// TIA Portal project "TankFillingSystem_V16" (V16)

(* hardware
DEVICE "S71500/ET200MP station_1"  S7-1500 station
   slot 0: "Rail_0"  Rack  6ES7 590-1***0-0AA0
   slot 1: "Tank filling controller"  CPU 1511C-1 PN  6ES7 511-1CK01-0AB0  V2.8
      slot 3: "CPU display_1"  6ES7591-1AA00-0AA0
      slot 32768: "PROFINET interface_1"  X1
         slot 32769: "Port_1"  X1 P1
         slot 32770: "Port_2"  X1 P2
      slot 34817: "Virtual CP interface port_1"  Virtual CP interface port  Virtual CP interface port
*)

// ===== PLC "Tank filling controller"  CPU 1511C-1 PN =====

VAR_GLOBAL   // PLC tag table "Default tag table"
   "Manual_Start" AT %I0.0 : Bool;
   "Work" AT %M2.0 : Bool;
   "Low_Level_Sensor" AT %I0.1 : Bool;
   "Low_Level" AT %M2.1 : Bool;
   "High_Level" AT %M2.2 : Bool;
   "Top_Level_Sensor" AT %I0.2 : Bool;
   "Manual_Stop" AT %I0.7 : Bool;
   "Manual_Valve_Control" AT %I0.3 : Bool;
   "Valve_Open" AT %M2.3 : Bool;
   "Tag_1" AT %I1.1 : Bool;
   "Manual_Confirm" AT %I0.6 : Bool;
   "Confirm" AT %M2.4 : Bool;
   "Clock_Byte" AT %MB50 : Byte;
   "Clock_10Hz" AT %M50.0 : Bool;
   "Clock_5Hz" AT %M50.1 : Bool;
   "Clock_2.5Hz" AT %M50.2 : Bool;
   "Clock_2Hz" AT %M50.3 : Bool;
   "Clock_1.25Hz" AT %M50.4 : Bool;
   "Clock_1Hz" AT %M50.5 : Bool;
   "Clock_0.625Hz" AT %M50.6 : Bool;
   "Clock_0.5Hz" AT %M50.7 : Bool;
   "Liquid_Montion_Sim" AT %M30.0 : Bool;
   "Emergency_Channel_Gen_Edge" AT %M2.5 : Bool;
   "Malfunction_Memory" AT %M2.6 : Bool;
   "Emergency_Channel_Malfunction_Edge" AT %M2.7 : Bool;
END_VAR

DATA_BLOCK "Tank1_DB"   // DB1
{ S7_Optimized_Access := 'TRUE' }
VERSION : 0.1
// stored: InstanceOfName Tank
"Tank"
BEGIN
   Capacity := 1000.0;
   Fill_Level := 1000.0;
   Growth := 2.5;
END_DATA_BLOCK

DATA_BLOCK "Pump_DB"   // DB2
{ S7_Optimized_Access := 'TRUE' }
VERSION : 0.1
// stored: InstanceOfName Pump
"Pump"
BEGIN
   Growth := 2.5;
END_DATA_BLOCK

DATA_BLOCK "RemoteControl"   // DB3
{ S7_Optimized_Access := 'TRUE' }
VERSION : 0.1
   VAR
      Start_Remote : Bool;
      Stop_Remote : Bool;
      Low_Level_Sensor_Remote : Bool;
      High_Level_Sensor_Remote : Bool;
      Valve_Control_Remote : Bool;
      Malfunction_Confirm_Remote : Bool;
      WWW_Return : Byte;
   END_VAR
BEGIN
END_DATA_BLOCK

DATA_BLOCK "ProcessControl"   // DB4
{ S7_Optimized_Access := 'TRUE' }
VERSION : 0.1
   VAR
      Fluid_at_Low_Level : Bool;
      Fluid_at_High_Level : Bool;
      Tank_Malfunction : Bool;
      Valve_Status : Bool;
      Pump_Work : Bool;
   END_VAR
BEGIN
END_DATA_BLOCK

FUNCTION_BLOCK "Tank"   // FB1, LAD
TITLE = Tank
{ S7_Optimized_Access := 'TRUE' }
VERSION : 0.1
// The logic for signalization of liquid level in the tank
   VAR_INPUT
      Botom_Level_Sensor : Bool;   // Bottom level sensor reading
      Top_Level_Sensor : Bool;   // Top level sensor reading
      Valve_Control : Bool;   // Valve control - open / close
   END_VAR
   VAR_OUTPUT
      Low_Level : Bool;   // The liquid is at the low level in tank
      High_Level : Bool;   // The liquid is at the high level in tank
      Malfunction : Bool;   // Malfunction: tank is leaning
      Valve_Status : Bool;   // Output infromation about valve status is open or closed
   END_VAR
   VAR
      Capacity : Real;   // Tank capacity
      Fill_Level : Real;   // Current fill level of liquid
      Valve_Remote : Bool;   // Valve remote controlling
      Generator_Edge : Bool;
      Growth : Real;   // how fill level decrease
   END_VAR
   VAR_TEMP   // added for the SCL form of the ladder/FBD networks
      _w1 : Bool;
   END_VAR
BEGIN

REGION Network 1: the liquid is at the low level in tank
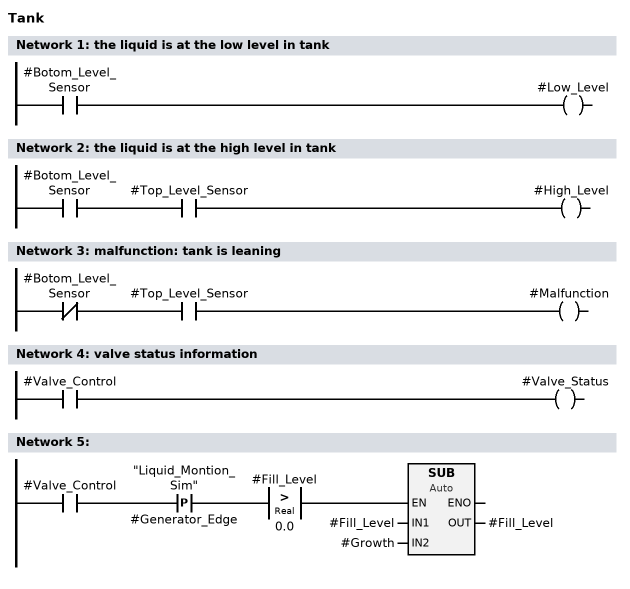
   RUNG wire#powerrail
      Contact( #Botom_Level_Sensor )
      Coil( #Low_Level )
   END_RUNG
   // the same network as SCL:
   #Low_Level := #Botom_Level_Sensor;
END_REGION

REGION Network 2: the liquid is at the high level in tank
   RUNG wire#powerrail
      Contact( #Botom_Level_Sensor )
      Contact( #Top_Level_Sensor )
      Coil( #High_Level )
   END_RUNG
   // the same network as SCL:
   #High_Level := #Botom_Level_Sensor AND #Top_Level_Sensor;
END_REGION

REGION Network 3: malfunction: tank is leaning
   RUNG wire#powerrail
      I_Contact( #Botom_Level_Sensor )
      Contact( #Top_Level_Sensor )
      Coil( #Malfunction )
   END_RUNG
   // the same network as SCL:
   #Malfunction := NOT #Botom_Level_Sensor AND #Top_Level_Sensor;
END_REGION

REGION Network 4: valve status information
   RUNG wire#powerrail
      Contact( #Valve_Control )
      Coil( #Valve_Status )
   END_RUNG
   // the same network as SCL:
   #Valve_Status := #Valve_Control;
END_REGION

REGION Network 5
   RUNG wire#powerrail
      Contact( #Valve_Control )
      P_Contact(operand := "Liquid_Montion_Sim", bit := #Generator_Edge)
      { S7_Templates := "SrcType := Real" } GT_Contact(in1 := #Fill_Level, in2 := 0.0)
      Sub(in1 := #Fill_Level, in2 := #Growth, out => #Fill_Level)
   END_RUNG
   // the same network as SCL:
   #_w1 := #Valve_Control AND "Liquid_Montion_Sim" AND NOT #Generator_Edge;   // rising edge of "Liquid_Montion_Sim"
   #Generator_Edge := "Liquid_Montion_Sim";
   IF #_w1 AND (#Fill_Level > 0.0) THEN #Fill_Level := #Fill_Level - #Growth; END_IF;
END_REGION
END_FUNCTION_BLOCK

FUNCTION_BLOCK "Pump"   // FB2, LAD
TITLE = Pump
{ S7_Optimized_Access := 'TRUE' }
VERSION : 0.1
// Logic of pump controlling
   VAR_INPUT
      Low_Level : Bool;   // Liquid level is at low
      Top_Level : Bool;   // Liquid level is at top
      Malfunction : Bool;   // Tank malfunction input information
      Capacity : Real;   // Tank capacity
   END_VAR
   VAR_OUTPUT
      Work_Status : Bool;   // pump is working
   END_VAR
   VAR_IN_OUT
      FillLevel : Real;
   END_VAR
   VAR
      Growth : Real;   // value of fill level increase
      Work : Bool;
      Generator_Edge : Bool;
   END_VAR
   VAR_TEMP   // added for the SCL form of the ladder/FBD networks
      _w1 : Bool;
   END_VAR
BEGIN

REGION Network 1: pump is working
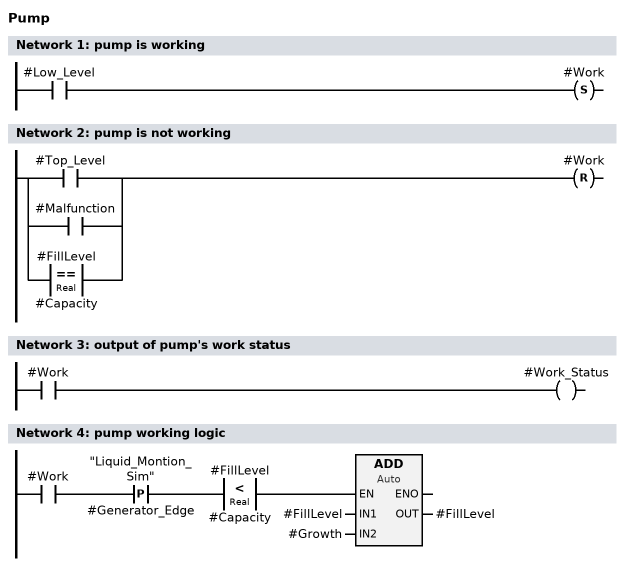
   RUNG wire#powerrail
      Contact( #Low_Level )
      S_Coil( #Work )
   END_RUNG
   // the same network as SCL:
   IF #Low_Level THEN #Work := TRUE; END_IF;
END_REGION

REGION Network 2: pump is not working
   RUNG wire#powerrail
      Contact( #Top_Level )
      wire#w1
      R_Coil( #Work )
   END_RUNG
   RUNG wire#powerrail
      Contact( #Malfunction )
   END_RUNG wire#w1
   RUNG wire#powerrail
      { S7_Templates := "SrcType := Real" } EQ_Contact(in1 := #FillLevel, in2 := #Capacity)
   END_RUNG wire#w1
   // the same network as SCL:
   IF #Top_Level OR #Malfunction OR (#FillLevel = #Capacity) THEN #Work := FALSE; END_IF;
END_REGION

REGION Network 3: output of pump's work status
   RUNG wire#powerrail
      Contact( #Work )
      Coil( #Work_Status )
   END_RUNG
   // the same network as SCL:
   #Work_Status := #Work;
END_REGION

REGION Network 4: pump working logic
   RUNG wire#powerrail
      Contact( #Work )
      P_Contact(operand := "Liquid_Montion_Sim", bit := #Generator_Edge)
      { S7_Templates := "SrcType := Real" } LT_Contact(in1 := #FillLevel, in2 := #Capacity)
      Add(in1 := #FillLevel, in2 := #Growth, out => #FillLevel)
   END_RUNG
   // the same network as SCL:
   #_w1 := #Work AND "Liquid_Montion_Sim" AND NOT #Generator_Edge;   // rising edge of "Liquid_Montion_Sim"
   #Generator_Edge := "Liquid_Montion_Sim";
   IF #_w1 AND (#FillLevel < #Capacity) THEN #FillLevel := #FillLevel + #Growth; END_IF;
END_REGION
END_FUNCTION_BLOCK

FUNCTION "EmergencyChannel" : Void   // FC1, LAD
{ S7_Optimized_Access := 'TRUE' }
VERSION : 0.1
   VAR_INPUT
      Hardware_Generator : Bool;   // Hardware Generator for flashing sygnalization
      Confirm : Bool;   // Malfunction confirming
      Malfunction : Bool;   // information about occured malfunction
   END_VAR
   VAR_OUTPUT
      Malfunction_Signal : Bool;   // the signalization of occured malfunction: flashing, continous
   END_VAR
   VAR_IN_OUT
      Generator_Edge : Bool;   // Hardware Generator edge memory
      Malfunction_Memory : Bool;   // memory that store information about malfunction in the previous circle
      Malfunction_Edge : Bool;   // The Rising edge for malfunction input signal
   END_VAR
   VAR_TEMP   // added for the SCL form of the ladder/FBD networks
      _w1 : Bool;
   END_VAR
BEGIN

REGION Network 1: memory that store information about malfunction in the previous circle
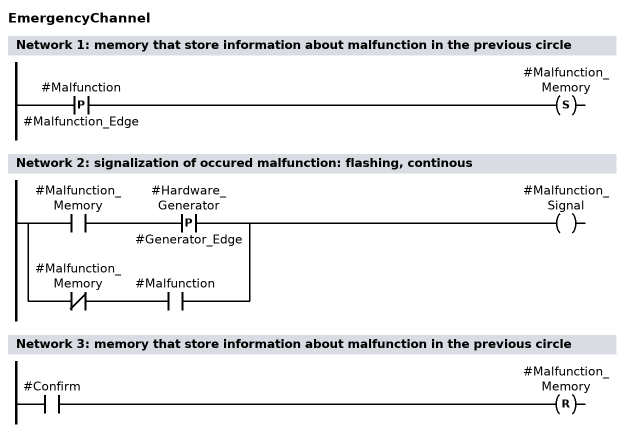
   RUNG wire#powerrail
      P_Contact(operand := #Malfunction, bit := #Malfunction_Edge)
      S_Coil( #Malfunction_Memory )
   END_RUNG
   // the same network as SCL:
   #_w1 := #Malfunction AND NOT #Malfunction_Edge;   // rising edge of #Malfunction
   #Malfunction_Edge := #Malfunction;
   IF #_w1 THEN #Malfunction_Memory := TRUE; END_IF;
END_REGION

REGION Network 2: signalization of occured malfunction: flashing, continous
   RUNG wire#powerrail
      Contact( #Malfunction_Memory )
      P_Contact(operand := #Hardware_Generator, bit := #Generator_Edge)
      wire#w1
      Coil( #Malfunction_Signal )
   END_RUNG
   RUNG wire#powerrail
      I_Contact( #Malfunction_Memory )
      Contact( #Malfunction )
   END_RUNG wire#w1
   // the same network as SCL:
   #_w1 := #Malfunction_Memory AND #Hardware_Generator AND NOT #Generator_Edge;   // rising edge of #Hardware_Generator
   #Generator_Edge := #Hardware_Generator;
   #Malfunction_Signal := #_w1 OR (NOT #Malfunction_Memory AND #Malfunction);
END_REGION

REGION Network 3: memory that store information about malfunction in the previous circle
   RUNG wire#powerrail
      Contact( #Confirm )
      R_Coil( #Malfunction_Memory )
   END_RUNG
   // the same network as SCL:
   IF #Confirm THEN #Malfunction_Memory := FALSE; END_IF;
END_REGION
END_FUNCTION

ORGANIZATION_BLOCK "Main"   // OB1, LAD, ProgramCycle
TITLE = "Main Program Sweep (Cycle)"
{ S7_Optimized_Access := 'TRUE' }
VERSION : 0.1
   VAR_INPUT
      Initial_Call : Bool;   // Initial call of this OB
      Remanence : Bool;   // =True, if remanent data are available
   END_VAR
BEGIN

REGION Network 1
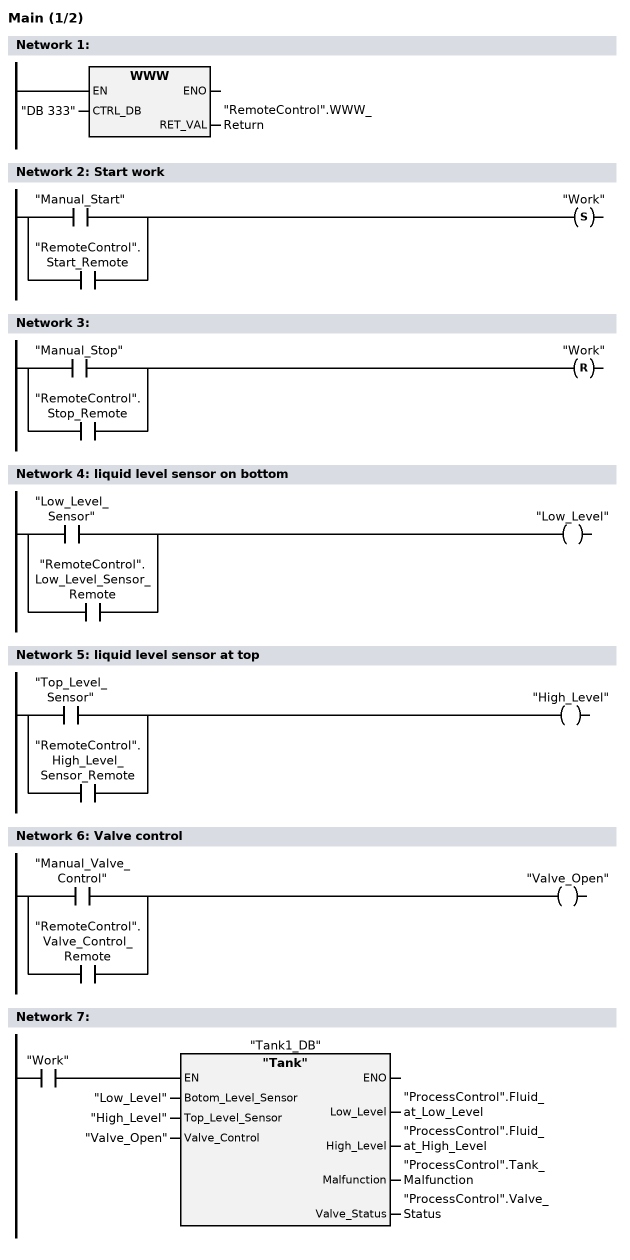
   "RemoteControl".WWW_Return := WWW(CTRL_DB := "DB 333");
END_REGION

REGION Network 2: Start work
   RUNG wire#powerrail
      Contact( "Manual_Start" )
      wire#w1
      S_Coil( "Work" )
   END_RUNG
   RUNG wire#powerrail
      Contact( "RemoteControl".Start_Remote )
   END_RUNG wire#w1
   // the same network as SCL:
   IF "Manual_Start" OR "RemoteControl".Start_Remote THEN "Work" := TRUE; END_IF;
END_REGION

REGION Network 3
   RUNG wire#powerrail
      Contact( "Manual_Stop" )
      wire#w1
      R_Coil( "Work" )
   END_RUNG
   RUNG wire#powerrail
      Contact( "RemoteControl".Stop_Remote )
   END_RUNG wire#w1
   // the same network as SCL:
   IF "Manual_Stop" OR "RemoteControl".Stop_Remote THEN "Work" := FALSE; END_IF;
END_REGION

REGION Network 4: liquid level sensor on bottom
   RUNG wire#powerrail
      Contact( "Low_Level_Sensor" )
      wire#w1
      Coil( "Low_Level" )
   END_RUNG
   RUNG wire#powerrail
      Contact( "RemoteControl".Low_Level_Sensor_Remote )
   END_RUNG wire#w1
   // the same network as SCL:
   "Low_Level" := "Low_Level_Sensor" OR "RemoteControl".Low_Level_Sensor_Remote;
END_REGION

REGION Network 5: liquid level sensor at top
   RUNG wire#powerrail
      Contact( "Top_Level_Sensor" )
      wire#w1
      Coil( "High_Level" )
   END_RUNG
   RUNG wire#powerrail
      Contact( "RemoteControl".High_Level_Sensor_Remote )
   END_RUNG wire#w1
   // the same network as SCL:
   "High_Level" := "Top_Level_Sensor" OR "RemoteControl".High_Level_Sensor_Remote;
END_REGION

REGION Network 6: Valve control
   RUNG wire#powerrail
      Contact( "Manual_Valve_Control" )
      wire#w1
      Coil( "Valve_Open" )
   END_RUNG
   RUNG wire#powerrail
      Contact( "RemoteControl".Valve_Control_Remote )
   END_RUNG wire#w1
   // the same network as SCL:
   "Valve_Open" := "Manual_Valve_Control" OR "RemoteControl".Valve_Control_Remote;
END_REGION

REGION Network 7
   RUNG wire#powerrail
      Contact( "Work" )
      "Tank1_DB"(Botom_Level_Sensor := "Low_Level", Top_Level_Sensor := "High_Level", Valve_Control := "Valve_Open", Low_Level => "ProcessControl".Fluid_at_Low_Level, High_Level => "ProcessControl".Fluid_at_High_Level, Malfunction => "ProcessControl".Tank_Malfunction, Valve_Status => "ProcessControl".Valve_Status)
   END_RUNG
   // the same network as SCL:
   IF "Work" THEN
       "Tank1_DB"(Botom_Level_Sensor := "Low_Level",   // "Tank"
                  Top_Level_Sensor := "High_Level",
                  Valve_Control := "Valve_Open",
                  Low_Level => "ProcessControl".Fluid_at_Low_Level,
                  High_Level => "ProcessControl".Fluid_at_High_Level,
                  Malfunction => "ProcessControl".Tank_Malfunction,
                  Valve_Status => "ProcessControl".Valve_Status);
   END_IF;
END_REGION

REGION Network 8
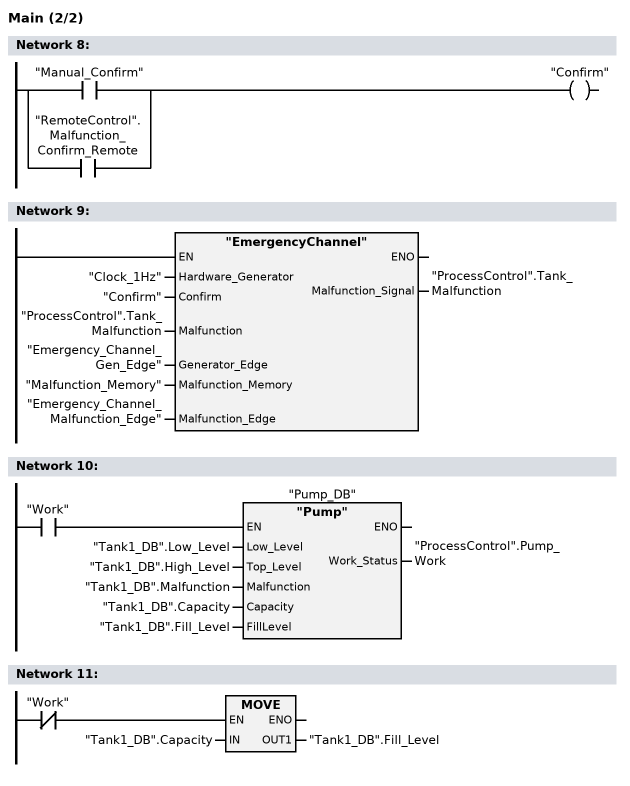
   RUNG wire#powerrail
      Contact( "Manual_Confirm" )
      wire#w1
      Coil( "Confirm" )
   END_RUNG
   RUNG wire#powerrail
      Contact( "RemoteControl".Malfunction_Confirm_Remote )
   END_RUNG wire#w1
   // the same network as SCL:
   "Confirm" := "Manual_Confirm" OR "RemoteControl".Malfunction_Confirm_Remote;
END_REGION

REGION Network 9
   RUNG wire#powerrail
      "EmergencyChannel"(Hardware_Generator := "Clock_1Hz", Confirm := "Confirm", Malfunction := "ProcessControl".Tank_Malfunction, Generator_Edge := "Emergency_Channel_Gen_Edge", Malfunction_Memory := "Malfunction_Memory", Malfunction_Edge := "Emergency_Channel_Malfunction_Edge", Malfunction_Signal => "ProcessControl".Tank_Malfunction)
   END_RUNG
   // the same network as SCL:
   "EmergencyChannel"(Hardware_Generator := "Clock_1Hz",
                      Confirm := "Confirm",
                      Malfunction := "ProcessControl".Tank_Malfunction,
                      Generator_Edge := "Emergency_Channel_Gen_Edge",
                      Malfunction_Memory := "Malfunction_Memory",
                      Malfunction_Edge := "Emergency_Channel_Malfunction_Edge",
                      Malfunction_Signal => "ProcessControl".Tank_Malfunction);
END_REGION

REGION Network 10
   RUNG wire#powerrail
      Contact( "Work" )
      "Pump_DB"(Low_Level := "Tank1_DB".Low_Level, Top_Level := "Tank1_DB".High_Level, Malfunction := "Tank1_DB".Malfunction, Capacity := "Tank1_DB".Capacity, FillLevel := "Tank1_DB".Fill_Level, Work_Status => "ProcessControl".Pump_Work)
   END_RUNG
   // the same network as SCL:
   IF "Work" THEN
       "Pump_DB"(Low_Level := "Tank1_DB".Low_Level,   // "Pump"
                 Top_Level := "Tank1_DB".High_Level,
                 Malfunction := "Tank1_DB".Malfunction,
                 Capacity := "Tank1_DB".Capacity,
                 FillLevel := "Tank1_DB".Fill_Level,
                 Work_Status => "ProcessControl".Pump_Work);
   END_IF;
END_REGION

REGION Network 11
   RUNG wire#powerrail
      I_Contact( "Work" )
      Move(in := "Tank1_DB".Capacity, out1 => "Tank1_DB".Fill_Level)
   END_RUNG
   // the same network as SCL:
   IF NOT "Work" THEN "Tank1_DB".Fill_Level := "Tank1_DB".Capacity; END_IF;
END_REGION
END_ORGANIZATION_BLOCK

ORGANIZATION_BLOCK "Liquid_Montion"   // OB30, LAD, CyclicInterrupt
{ S7_Optimized_Access := 'TRUE' }
VERSION : 0.1
   VAR_INPUT
      Initial_Call : Bool;   // Initial call of this OB
      Event_Count : Int;   // Events discarded
   END_VAR
BEGIN

REGION Network 1
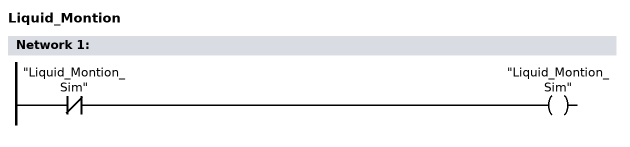
   RUNG wire#powerrail
      I_Contact( "Liquid_Montion_Sim" )
      Coil( "Liquid_Montion_Sim" )
   END_RUNG
   // the same network as SCL:
   "Liquid_Montion_Sim" := NOT "Liquid_Montion_Sim";
END_REGION
END_ORGANIZATION_BLOCK

ORGANIZATION_BLOCK "Startup"   // OB100, LAD, Startup
TITLE = "Complete Restart"
{ S7_Optimized_Access := 'TRUE' }
VERSION : 0.1
   VAR_INPUT
      LostRetentive : Bool;   // True if retentive data are lost
      LostRTC : Bool;   // True if date and time are lost
   END_VAR
BEGIN

REGION Network 1
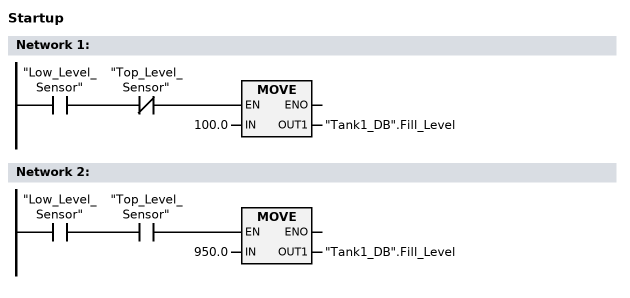
   RUNG wire#powerrail
      Contact( "Low_Level_Sensor" )
      I_Contact( "Top_Level_Sensor" )
      Move(in := 100.0, out1 => "Tank1_DB".Fill_Level)
   END_RUNG
   // the same network as SCL:
   IF "Low_Level_Sensor" AND NOT "Top_Level_Sensor" THEN "Tank1_DB".Fill_Level := 100.0; END_IF;
END_REGION

REGION Network 2
   RUNG wire#powerrail
      Contact( "Low_Level_Sensor" )
      Contact( "Top_Level_Sensor" )
      Move(in := 950.0, out1 => "Tank1_DB".Fill_Level)
   END_RUNG
   // the same network as SCL:
   IF "Low_Level_Sensor" AND "Top_Level_Sensor" THEN "Tank1_DB".Fill_Level := 950.0; END_IF;
END_REGION
END_ORGANIZATION_BLOCK